(*udt (user defined type) Device Info Data Section (configurable) of Beckhoff EL6900 - TwinSAFE Controller
	auth. Brent Lekx-Toniolo of Sodecia GTAC.; 
------------------------------------------------------------------------
REVISION NOTES:
	Version 20160426
			- Original Concept, b.lekx-toniolo

------------------------------------------------------------------------

*)



TYPE udt_EL6900_DeviceInfoData_20160426 :
	STRUCT
		(*Project CRC*)
		Project_CRC: UINT;

	END_STRUCT
END_TYPE

(* stored: Version 1.1.0.1, ProductVersion 3.1.4024.9
   DUT udt_EL6900_DeviceInfoData_20160426: Id {f1ee9d8e-4485-42e5-a866-d64d7ddd0b64} *)
